# EPICS autosave request: iocBoot/generic_motors_ioc/dbSave/mtr1.req
%
% BURT Request File
%
% MOTOR
%

% RO $(MTR1):ActPos
$(MTR1):ActPos.EGU
$(MTR1):ActPos.DESC

$(MTR1):RqsPos
$(MTR1):RqsPos.EGU
$(MTR1):RqsPos.DESC
$(MTR1):RqsPos.HOPR
$(MTR1):RqsPos.LOPR
$(MTR1):RqsPos.DRVH
$(MTR1):RqsPos.DRVL

$(MTR1):RqsBkl
$(MTR1):RqsBkl.EGU
$(MTR1):RqsBkl.DESC

$(MTR1):RqsPosInc
$(MTR1):MemPos
